// Mitsubishi GX Works2 project: PressureRead   PLC: FX3U/FX3UC

PROGRAM MAIN
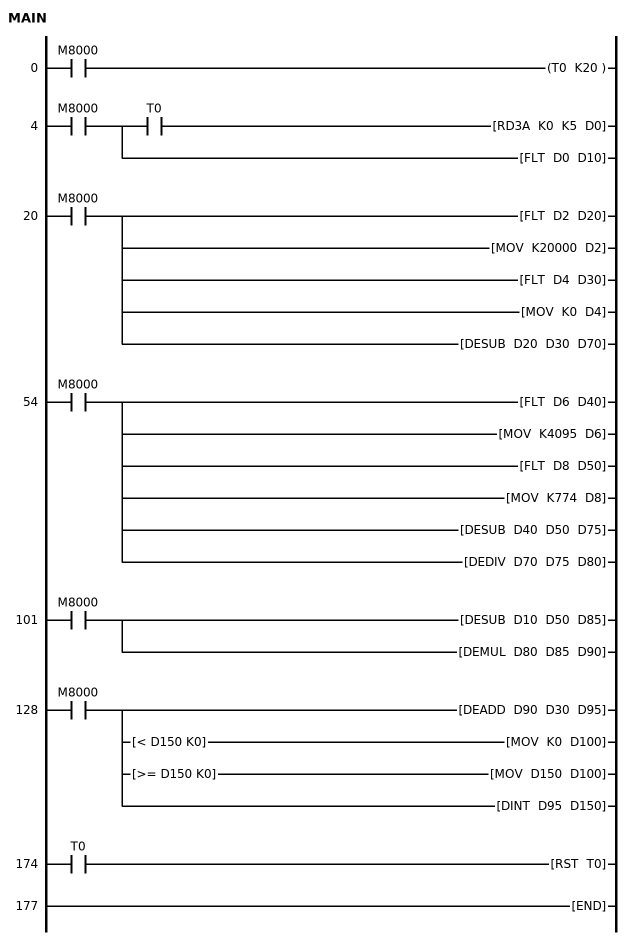
0     LD      M8000
      OUT     T0 K20
4     LD      M8000
      MPS
      AND     T0
      RD3A    K0 K5 D0
      MPP
      FLT     D0 D10
20    LD      M8000
      FLT     D2 D20
      MOV     K20000 D2
      FLT     D4 D30
      MOV     K0 D4
      DESUB   D20 D30 D70
54    LD      M8000
      FLT     D6 D40
      MOV     K4095 D6
      FLT     D8 D50
      MOV     K774 D8
      DESUB   D40 D50 D75
      DEDIV   D70 D75 D80
101   LD      M8000
      DESUB   D10 D50 D85
      DEMUL   D80 D85 D90
128   LD      M8000
      DEADD   D90 D30 D95
      MPS
      AND<    D150 K0
      MOV     K0 D100
      MRD
      AND>=   D150 K0
      MOV     D150 D100
      MPP
      DINT    D95 D150
174   LD      T0
      RST     T0
177   END
END_PROGRAM
